// TIA Portal V15.1 export
// export: Created 2024-05-17T05:38:44.1667821Z, ExportSetting WithDefaults, DisplayName Totally Integrated Automation Portal, DisplayVersion V15.1 Update 5, DisplayName TIA Portal Openness, DisplayVersion V15.1 Update 5, DisplayName SINAMICS Startdrive Advanced, DisplayVersion V15.1, DisplayName G130, G150, S120, S150, SINAMICS MV, S210, DisplayVersion V15.1, DisplayName G110M, G120, G120C, G120D, G120P, DisplayVersion V15.1, DisplayName STEP 7 Professional, DisplayVersion V15.1 Update 5, DisplayName STEP 7 Safety, DisplayVersion V15.1, DisplayName WinCC Professional, DisplayVersion V15.1 Update 5, DisplayName SIMATIC Visualization Architect, DisplayVersion V15.1
FUNCTION_BLOCK "LGBVIDSChangeVEMData"   // FB6633, SCL
TITLE = LGBVIDSChangeVEMData
{ S7_Optimized_Access := 'FALSE' }
VERSION : 0.1
// stored: AutoNumber false, IsIECCheckEnabled false, SetENOAutomatically False, UDAEnableTagReadback false
   VAR_INPUT
      I_StartChangeVEMData { ExternalAccessible := 'False'; ExternalVisible := 'False'; ExternalWritable := 'False'} : Bool;   // Start command for coupling / Start command
      I_DataModeManEn { ExternalAccessible := 'False'; ExternalVisible := 'False'; ExternalWritable := 'False'} : Bool;   // Data mode manual - enable
   END_VAR
   VAR_OUTPUT
      O_DataModeAuto { ExternalAccessible := 'False'; ExternalVisible := 'False'; ExternalWritable := 'False'} : Bool;   // Couple or decouple in automatic mode / Data mode - Automatic
      O_DataModeMan { ExternalAccessible := 'False'; ExternalVisible := 'False'; ExternalWritable := 'False'} : Bool;   // Data mode - Manual
      O_Busy { ExternalAccessible := 'False'; ExternalVisible := 'False'; ExternalWritable := 'False'} : Bool;   // Busy
      O_Status { ExternalAccessible := 'False'; ExternalVisible := 'False'; ExternalWritable := 'False'} : Int;   // Status / Status (< 0 : fault, 0:No status, 1:Success, >0:Busy)
      O_Alarm { ExternalAccessible := 'False'; ExternalVisible := 'False'; ExternalWritable := 'False'} : Bool;   // Alarm
   END_VAR
   VAR_IN_OUT
      IO_VIDS : "VIDS";   // VIDS internal record
      IO_VEMData : "VEMData";   // VEM data
      IO_VEMDataChange : "VEMData";   // VEM data to be changed
      IO_CarrierCargoStatus : "VIDSCarrierCargoStatus";   // Carrier cargo status (Fixed layout)
      IO_CarrierCargoStatusChange : "VIDSCarrierCargoStatus";   // Carrier cargo status to be changed(Fixed layout)
      IO_BodyCargoStatus : "VIDSBodyCargoStatusGB";   // Body cargo status (Fixed layout)
      IO_BodyCargoStatusChange : "VIDSBodyCargoStatusGB";   // Body cargo status to be changed(Fixed layout)
      IO_WorkStatus : "VIDSWorkStatus";   // Work status(Fixed layout)
      IO_WorkStatusChange : "VIDSWorkStatus";   // Work status to be changed(Fixed layout)
      IO_EquipmentWork : "VIDSEquipment";
      IO_EquipmentWorkChange : "VIDSEquipment";
      IO_EquipmentWorkDone : "VIDSEquipment";
      IO_EquipmentWorkDoneChange : "VIDSEquipment";
      IO_Alarm : "Alarm";   // Alarm
      H_ChangeVEMData : "H_GBVIDSChangeVEMData";   // HMI interface
      H_HMI : "H_HMI";   // Icon animation
   END_VAR
   VAR DB_SPECIFIC
      RetVal { ExternalAccessible := 'False'; ExternalVisible := 'False'; ExternalWritable := 'False'} : Int;
      StartChangeVEMDataPls { ExternalAccessible := 'False'; ExternalVisible := 'False'; ExternalWritable := 'False'} : Bool;
      btnConfirmPls { ExternalAccessible := 'False'; ExternalVisible := 'False'; ExternalWritable := 'False'} : Bool;
      btnEditPls { ExternalAccessible := 'False'; ExternalVisible := 'False'; ExternalWritable := 'False'} : Bool;
      DataModeAuto { ExternalAccessible := 'False'; ExternalVisible := 'False'; ExternalWritable := 'False'} : Bool;   // Couple or decouple in automode
      DataModeAutoPls { ExternalAccessible := 'False'; ExternalVisible := 'False'; ExternalWritable := 'False'} : Bool;
      DataModeMan { ExternalAccessible := 'False'; ExternalVisible := 'False'; ExternalWritable := 'False'} : Bool;
      DataModeManPls { ExternalAccessible := 'False'; ExternalVisible := 'False'; ExternalWritable := 'False'} : Bool;
      DataModeMem { ExternalAccessible := 'False'; ExternalVisible := 'False'; ExternalWritable := 'False'} : Int;
      DataModeEdit { ExternalAccessible := 'False'; ExternalVisible := 'False'; ExternalWritable := 'False'} : Bool;
      DataModeChanged { ExternalAccessible := 'False'; ExternalVisible := 'False'; ExternalWritable := 'False'} : Bool;
      BeginReqPlsAuto { ExternalAccessible := 'False'; ExternalVisible := 'False'; ExternalWritable := 'False'} : Bool;
      BeginReqPlsMan { ExternalAccessible := 'False'; ExternalVisible := 'False'; ExternalWritable := 'False'} : Bool;
      SerializePos { ExternalAccessible := 'False'; ExternalVisible := 'False'; ExternalWritable := 'False'} : DInt;
      DeSerializePos { ExternalAccessible := 'False'; ExternalVisible := 'False'; ExternalWritable := 'False'} : DInt;
      VEMDataChangeMem { ExternalAccessible := 'False'; ExternalVisible := 'False'; ExternalWritable := 'False'; S7_SetPoint := 'True'} : "VEMData";
      VEMDataChangeMemArray { ExternalAccessible := 'False'; ExternalVisible := 'False'; ExternalWritable := 'False'} : Array[0..255] of Byte;
      Busy { ExternalAccessible := 'False'; ExternalVisible := 'False'; ExternalWritable := 'False'} : Bool;
      btnDataModeAutoColour { ExternalAccessible := 'False'; ExternalVisible := 'False'; ExternalWritable := 'False'} : Word;
      btnDataModeManColour { ExternalAccessible := 'False'; ExternalVisible := 'False'; ExternalWritable := 'False'} : Word;
      CarrierID { ExternalAccessible := 'False'; ExternalVisible := 'False'; ExternalWritable := 'False'} : DWord;
      CarrierIDValid { ExternalAccessible := 'False'; ExternalVisible := 'False'; ExternalWritable := 'False'} : Bool;
      CarrierIDMem { ExternalAccessible := 'False'; ExternalVisible := 'False'; ExternalWritable := 'False'} : DWord;   // Memory of CarrierID at begin request
      TagID { ExternalAccessible := 'False'; ExternalVisible := 'False'; ExternalWritable := 'False'} : DWord;
      TagIDValid { ExternalAccessible := 'False'; ExternalVisible := 'False'; ExternalWritable := 'False'} : Bool;
      TagIDMem { ExternalAccessible := 'False'; ExternalVisible := 'False'; ExternalWritable := 'False'} : DWord;
      BodyNbr { ExternalAccessible := 'False'; ExternalVisible := 'False'; ExternalWritable := 'False'} : DWord;
      BodyNbrValid { ExternalAccessible := 'False'; ExternalVisible := 'False'; ExternalWritable := 'False'} : Bool;
      BodyNbrMem { ExternalAccessible := 'False'; ExternalVisible := 'False'; ExternalWritable := 'False'} : DWord;
      MixNbr { ExternalAccessible := 'False'; ExternalVisible := 'False'; ExternalWritable := 'False'} : DWord;
      MixNbrValid { ExternalAccessible := 'False'; ExternalVisible := 'False'; ExternalWritable := 'False'} : Bool;
      MixNbrMem { ExternalAccessible := 'False'; ExternalVisible := 'False'; ExternalWritable := 'False'} : DWord;
      DataValid { ExternalAccessible := 'False'; ExternalVisible := 'False'; ExternalWritable := 'False'} : Bool;
      VEMDataValidPls { ExternalAccessible := 'False'; ExternalVisible := 'False'; ExternalWritable := 'False'} : Bool;
      InputDataValidAuto { ExternalAccessible := 'False'; ExternalVisible := 'False'; ExternalWritable := 'False'} : Bool;
      InputDataValidMan { ExternalAccessible := 'False'; ExternalVisible := 'False'; ExternalWritable := 'False'} : Bool;
      DataNotValid { ExternalAccessible := 'False'; ExternalVisible := 'False'; ExternalWritable := 'False'} : Bool;
      BeginPlsModeAuto { ExternalAccessible := 'False'; ExternalVisible := 'False'; ExternalWritable := 'False'} : Bool;   // Pulse of begin in auto mode
      BeginPlsModeManTagId { ExternalAccessible := 'False'; ExternalVisible := 'False'; ExternalWritable := 'False'} : Bool;   // Pulse of begin in manual mode
      BeginReqPls { ExternalAccessible := 'False'; ExternalVisible := 'False'; ExternalWritable := 'False'} : Bool;   // Pulse of begin request
      TagIdModeManMem { ExternalAccessible := 'False'; ExternalVisible := 'False'; ExternalWritable := 'False'} : DWord;   // Memorised TagId in manual mode
      Alarm { ExternalAccessible := 'False'; ExternalVisible := 'False'; ExternalWritable := 'False'} : Bool;   // Alarm
      ChangedRcvDataAlarm { ExternalAccessible := 'False'; ExternalVisible := 'False'; ExternalWritable := 'False'} : Bool;   // Alarm received data has chnged after request
      CoupleAlarm { ExternalAccessible := 'False'; ExternalVisible := 'False'; ExternalWritable := 'False'} : Bool;   // Alarm couple or decouple NOK
      Status { ExternalAccessible := 'False'; ExternalVisible := 'False'; ExternalWritable := 'False'} : Int;   // Status
      btnEditVisible { ExternalAccessible := 'False'; ExternalVisible := 'False'; ExternalWritable := 'False'} : Word;
      btnEditEnable { ExternalAccessible := 'False'; ExternalVisible := 'False'; ExternalWritable := 'False'} : Word;
      btnConfirmVisible { ExternalAccessible := 'False'; ExternalVisible := 'False'; ExternalWritable := 'False'} : Word;
      btnConfirmEnable { ExternalAccessible := 'False'; ExternalVisible := 'False'; ExternalWritable := 'False'} : Word;
      msgDataValidVisible { ExternalAccessible := 'False'; ExternalVisible := 'False'; ExternalWritable := 'False'} : Word;   // HMI - Couple/Decouple OK
      msgDataNotValidVisible { ExternalAccessible := 'False'; ExternalVisible := 'False'; ExternalWritable := 'False'} : Word;   // HMI - Couple/Decouple OK
      msgPartPresVisible { ExternalAccessible := 'False'; ExternalVisible := 'False'; ExternalWritable := 'False'} : Word;
      msgVEMDataCarrierVisible { ExternalAccessible := 'False'; ExternalVisible := 'False'; ExternalWritable := 'False'} : Word;
      msgVEMDataBodyVisible { ExternalAccessible := 'False'; ExternalVisible := 'False'; ExternalWritable := 'False'} : Word;
      txtCarrierIDVisible { ExternalAccessible := 'False'; ExternalVisible := 'False'; ExternalWritable := 'False'} : Word;
      txtCarrierIDEnable { ExternalAccessible := 'False'; ExternalVisible := 'False'; ExternalWritable := 'False'} : Word;
      txtCarrierIDColour { ExternalAccessible := 'False'; ExternalVisible := 'False'; ExternalWritable := 'False'} : Word;
      txtCarrierIDValid { ExternalAccessible := 'False'; ExternalVisible := 'False'; ExternalWritable := 'False'} : Bool;
      txtTagIDVisible { ExternalAccessible := 'False'; ExternalVisible := 'False'; ExternalWritable := 'False'} : Word;
      txtTagIDEnable { ExternalAccessible := 'False'; ExternalVisible := 'False'; ExternalWritable := 'False'} : Word;
      txtTagIDColour { ExternalAccessible := 'False'; ExternalVisible := 'False'; ExternalWritable := 'False'} : Word;
      txtTagIDValid { ExternalAccessible := 'False'; ExternalVisible := 'False'; ExternalWritable := 'False'} : Bool;
      txtMixNbrVisible { ExternalAccessible := 'False'; ExternalVisible := 'False'; ExternalWritable := 'False'} : Word;
      txtMixNbrEnable { ExternalAccessible := 'False'; ExternalVisible := 'False'; ExternalWritable := 'False'} : Word;
      txtMixNbrColour { ExternalAccessible := 'False'; ExternalVisible := 'False'; ExternalWritable := 'False'} : Word;
      txtMixNbrValid { ExternalAccessible := 'False'; ExternalVisible := 'False'; ExternalWritable := 'False'} : Bool;
      txtdestinationChangeVisible { ExternalAccessible := 'False'; ExternalVisible := 'False'; ExternalWritable := 'False'} : Word;
      txtdestinationChangeEnable { ExternalAccessible := 'False'; ExternalVisible := 'False'; ExternalWritable := 'False'} : Word;
      txtPlcProgramNumberChangeVisible { ExternalAccessible := 'False'; ExternalVisible := 'False'; ExternalWritable := 'False'} : Word;
      txtPlcProgramNumberChangeEnable { ExternalAccessible := 'False'; ExternalVisible := 'False'; ExternalWritable := 'False'} : Word;
      txtBodyNbrVisible { ExternalAccessible := 'False'; ExternalVisible := 'False'; ExternalWritable := 'False'} : Word;
      txtBodyNbrEnable { ExternalAccessible := 'False'; ExternalVisible := 'False'; ExternalWritable := 'False'} : Word;
      txtBodyNbrColour { ExternalAccessible := 'False'; ExternalVisible := 'False'; ExternalWritable := 'False'} : Word;
      txtBodyNbrValid { ExternalAccessible := 'False'; ExternalVisible := 'False'; ExternalWritable := 'False'} : Bool;
      txtSeqNbrChangeVisible { ExternalAccessible := 'False'; ExternalVisible := 'False'; ExternalWritable := 'False'} : Word;
      txtSeqNbrChangeEnable { ExternalAccessible := 'False'; ExternalVisible := 'False'; ExternalWritable := 'False'} : Word;
      txtRoutingChangeVisible { ExternalAccessible := 'False'; ExternalVisible := 'False'; ExternalWritable := 'False'} : Word;
      txtRoutingChangeEnable { ExternalAccessible := 'False'; ExternalVisible := 'False'; ExternalWritable := 'False'} : Word;
      txtWorkUntilChangeVisible { ExternalAccessible := 'False'; ExternalVisible := 'False'; ExternalWritable := 'False'} : Word;
      txtWorkUntilChangeEnable { ExternalAccessible := 'False'; ExternalVisible := 'False'; ExternalWritable := 'False'} : Word;
      txtBegWorkAfterChangeVisible { ExternalAccessible := 'False'; ExternalVisible := 'False'; ExternalWritable := 'False'} : Word;
      txtBegWorkAfterChangeEnable { ExternalAccessible := 'False'; ExternalVisible := 'False'; ExternalWritable := 'False'} : Word;
      selBodyCargoStatusChangeVisible { ExternalAccessible := 'False'; ExternalVisible := 'False'; ExternalWritable := 'False'} : Word;
      selBodyCargoStatusChangeEnable { ExternalAccessible := 'False'; ExternalVisible := 'False'; ExternalWritable := 'False'} : Word;
      selCarrierCargoStatusChangeVisible { ExternalAccessible := 'False'; ExternalVisible := 'False'; ExternalWritable := 'False'} : Word;
      selCarrierCargoStatusChangeEnable { ExternalAccessible := 'False'; ExternalVisible := 'False'; ExternalWritable := 'False'} : Word;
      selWorkStatusChangeVisible { ExternalAccessible := 'False'; ExternalVisible := 'False'; ExternalWritable := 'False'} : Word;
      selWorkStatusChangeEnable { ExternalAccessible := 'False'; ExternalVisible := 'False'; ExternalWritable := 'False'} : Word;
      selEquipmentWorkVisible { ExternalAccessible := 'False'; ExternalVisible := 'False'; ExternalWritable := 'False'} : Word;
      selEquipmentWorkEnable { ExternalAccessible := 'False'; ExternalVisible := 'False'; ExternalWritable := 'False'} : Word;
      selEquipmentWorkDoneVisible { ExternalAccessible := 'False'; ExternalVisible := 'False'; ExternalWritable := 'False'} : Word;
      selEquipmentWorkDoneEnable { ExternalAccessible := 'False'; ExternalVisible := 'False'; ExternalWritable := 'False'} : Word;
      IconColour { ExternalAccessible := 'False'; ExternalVisible := 'False'; ExternalWritable := 'False'} : Word;
      tempDWORDArray { ExternalAccessible := 'False'; ExternalVisible := 'False'; ExternalWritable := 'False'} : Array[0..31] of Bool;
   END_VAR
   VAR
      _DataModeManPls { ExternalAccessible := 'False'; ExternalVisible := 'False'; ExternalWritable := 'False'; S7_SetPoint := 'True'} : R_TRIG;
      _DataModeAutoPls { ExternalAccessible := 'False'; ExternalVisible := 'False'; ExternalWritable := 'False'; S7_SetPoint := 'True'} : R_TRIG;
      _btnConfirmPls { ExternalAccessible := 'False'; ExternalVisible := 'False'; ExternalWritable := 'False'; S7_SetPoint := 'True'} : R_TRIG;
      _btnEditPls { ExternalAccessible := 'False'; ExternalVisible := 'False'; ExternalWritable := 'False'; S7_SetPoint := 'True'} : R_TRIG;
      _VEMDataValidPls { ExternalAccessible := 'False'; ExternalVisible := 'False'; ExternalWritable := 'False'; S7_SetPoint := 'True'} : R_TRIG;
      _StartChangeVEMDataPls { ExternalAccessible := 'False'; ExternalVisible := 'False'; ExternalWritable := 'False'; S7_SetPoint := 'True'} : R_TRIG;
   END_VAR
   VAR DB_SPECIFIC
      _CoupleBeginOvTime { ExternalAccessible := 'False'; ExternalVisible := 'False'; ExternalWritable := 'False'; S7_SetPoint := 'True'} : TOF_TIME;
   END_VAR
   VAR
      _CoupleBeginWaitDonePls { ExternalAccessible := 'False'; ExternalVisible := 'False'; ExternalWritable := 'False'; S7_SetPoint := 'True'} : F_TRIG;
   END_VAR
   VAR DB_SPECIFIC
      _DeoupleBeginOvTime { ExternalAccessible := 'False'; ExternalVisible := 'False'; ExternalWritable := 'False'; S7_SetPoint := 'True'} : TOF_TIME;
   END_VAR
   VAR
      _DecoupleBeginWaitDonePls { ExternalAccessible := 'False'; ExternalVisible := 'False'; ExternalWritable := 'False'; S7_SetPoint := 'True'} : F_TRIG;
   END_VAR
   VAR_TEMP
      tempBool : Bool;
   END_VAR
   VAR CONSTANT
      STATUS_OK : Int := 1;
      STATUS_COUPLE_REQ : Int := 107;
      STATUS_COUPLE_RUNNING : Int := 207;
      STATUS_DECOUPLE_REQ : Int := 108;
      STATUS_DECOUPLE_RUNNING : Int := 208;
      OFF : Word := 2#0000000000000000;
      ON : Word := 2#0000000000000001;
      VISIBLE : Word := 2#0000000000000001;
      ENABLE : Word := 2#0000000000000010;
      COLOUR_DEFAULT : Word := 2#0000000000000000;
      COLOUR_RED : Word := 2#0000000000010000;
      COLOUR_GREEN : Word := 2#0000000000100000;
      COLOUR_BLUE : Word := 2#0000000001000000;
      COLOUR_WHITE : Word := 2#0000000010000000;
      CMD_CHANGE_DATA : DWord := 2001;
   END_VAR
BEGIN
   (******************************************************************************************
    Changelog

       21W29D3 18:00H 
       - New module

    List of authors

       Company : Volvo Cars Gent
       Name    : Christophe Staal
       E-mail  : christophe.staal@volvocars.com
       Tel.    : +32 470 34 60 98

    Description

       This module allows to change VEM data commonly used in B-shop

    ******************************************************************************)

   //Start change VEM data - Create pulse on edge
   #_StartChangeVEMDataPls(CLK := #I_StartChangeVEMData,
                   Q => #StartChangeVEMDataPls);

   //Button Confirm - Create pulse on edge
   #_btnConfirmPls(CLK := #H_ChangeVEMData.H_btnConfirm=#ON,
                   Q => #btnConfirmPls);

   //Button Edit - Create pulse on edge
   #_btnEditPls(CLK := #H_ChangeVEMData.H_btnEdit = #ON,
                Q => #btnEditPls);

   #_VEMDataValidPls(CLK := #IO_VIDS.VEMDataValid,
                Q => #VEMDataValidPls);

   (******************************************************************************)
   (* Data mode - Automatic                                                      *)
   (******************************************************************************)

   //Data mode selected  - No mode, select auto
      IF (#H_ChangeVEMData.H_selDataMode < 1) OR (#H_ChangeVEMData.H_selDataMode > 3) OR NOT #IO_VIDS.PartPres OR NOT #I_DataModeManEn THEN
          #H_ChangeVEMData.H_selDataMode := 1;
   END_IF;

   #DataModeAuto := #H_ChangeVEMData.H_selDataMode = 1;

   (******************************************************************************)
   (* Data mode - Manual                                                         *)
   (******************************************************************************)

   //Data mode MANUAL
   #DataModeMan := (#H_ChangeVEMData.H_selDataMode = 2);

   //Data mode changed
   #DataModeChanged := #H_ChangeVEMData.H_selDataMode <> #DataModeMem;
   #DataModeMem := #H_ChangeVEMData.H_selDataMode;

   (******************************************************************************)
   (* Data mode - Edit                                                           *)
   (******************************************************************************)

   IF #DataModeMan AND #btnEditPls THEN
       #DataModeEdit := TRUE;
   END_IF;

   (******************************************************************************)
   (* Update on VEM data valid                                                   *)
   (******************************************************************************)

   //Body Cargo status - update
   "LDWordToBit"(I_DWord:=#IO_VEMData.BodyCargoStatus,
                 O_0=>#IO_BodyCargoStatus.OK,
                 O_1=>#IO_BodyCargoStatus.NOK,
                 O_2=>#IO_BodyCargoStatus.Production,
                 O_3=>#IO_BodyCargoStatus.Test,
                 O_4=>#IO_BodyCargoStatus.Measurement,
                 O_5=>#IO_BodyCargoStatus.Scrap,
                 O_6=>#tempBool,
                 O_7=>#tempBool,
                 O_8=>#IO_BodyCargoStatus.Inspection,
                 O_9=>#tempBool,
                 O_10=>#IO_BodyCargoStatus.NoPriorityFlowDecisionByPLC,
                 O_11=>#IO_BodyCargoStatus.BodyCanGoTo5thCrane,
                 O_12=>#IO_BodyCargoStatus.BodyMustGoTo5thCrane,
                 O_13=>#IO_BodyCargoStatus.BodyCanNotGoTo5thCrane,
                 O_14=>#tempBool,
                 O_15=>#tempBool,
                 O_16=>#tempBool,
                 O_17=>#tempBool,
                 O_18=>#tempBool,
                 O_19=>#tempBool,
                 O_20=>#IO_BodyCargoStatus.BodyBufferFull,
                 O_21=>#IO_BodyCargoStatus.OvenBodyTC1Oven1,
                 O_22=>#IO_BodyCargoStatus.OvenBodyTC1Oven2,
                 O_23=>#IO_BodyCargoStatus.OvenBodyTC2Oven1,
                 O_24=>#IO_BodyCargoStatus.OvenBodyTC2Oven2,
                 O_25=>#IO_BodyCargoStatus.TestBodyTC1,
                 O_26=>#IO_BodyCargoStatus.TestBodyTC2,
                 O_27=>#tempBool,
                 O_28=>#tempBool,
                 O_29=>#tempBool,
                 O_30=>#tempBool,
                 O_31=>#IO_BodyCargoStatus.ExitWaterTestBody);

   //Carrier Cargo status - update
   "LDWordToBit"(I_DWord := #IO_VEMData.CarrierCargoStatus,
                 O_0 => #IO_CarrierCargoStatus.OK,
                 O_1 => #IO_CarrierCargoStatus.NOK,
                 O_2 => #IO_CarrierCargoStatus.Test,
                 O_3 => #IO_CarrierCargoStatus.Maint,
                 O_4 => #IO_CarrierCargoStatus.PrevMaint,
                 O_5 => #IO_CarrierCargoStatus.Loaded,
                 O_6 => #IO_CarrierCargoStatus.Job1,
                 O_7 => #IO_CarrierCargoStatus.Job2,
                 O_8 => #IO_CarrierCargoStatus.Job3,
                 O_9 => #tempBool,
                 O_10 => #tempBool,
                 O_11 => #tempBool,
                 O_12 => #tempBool,
                 O_13 => #tempBool,
                 O_14 => #tempBool,
                 O_15 => #tempBool,
                 O_16 => #tempBool,
                 O_17 => #tempBool,
                 O_18 => #tempBool,
                 O_19 => #tempBool,
                 O_20 => #tempBool,
                 O_21 => #tempBool,
                 O_22 => #tempBool,
                 O_23 => #tempBool,
                 O_24 => #tempBool,
                 O_25 => #tempBool,
                 O_26 => #tempBool,
                 O_27 => #tempBool,
                 O_28 => #tempBool,
                 O_29 => #tempBool,
                 O_30 => #tempBool,
                 O_31 => #tempBool);

   //Work status - update
   "LDWordToBit"(I_DWord := #IO_VEMData.WorkStatus,
                 O_0 => #IO_WorkStatus.Work,
                 O_1 => #IO_WorkStatus.NoWork,
                 O_2 => #IO_WorkStatus.BackupWork,
                 O_3 => #IO_WorkStatus.StopBefore,
                 O_4 => #IO_WorkStatus.StopAfter,
                 O_5 => #IO_WorkStatus.Quality,
                 O_6 => #tempBool,
                 O_7 => #tempBool,
                 O_8 => #tempBool,
                 O_9 => #tempBool,
                 O_10 => #tempBool,
                 O_11 => #tempBool,
                 O_12 => #tempBool,
                 O_13 => #tempBool,
                 O_14 => #tempBool,
                 O_15 => #tempBool,
                 O_16 => #tempBool,
                 O_17 => #tempBool,
                 O_18 => #tempBool,
                 O_19 => #tempBool,
                 O_20 => #tempBool,
                 O_21 => #tempBool,
                 O_22 => #tempBool,
                 O_23 => #tempBool,
                 O_24 => #tempBool,
                 O_25 => #tempBool,
                 O_26 => #tempBool,
                 O_27 => #tempBool,
                 O_28 => #tempBool,
                 O_29 => #tempBool,
                 O_30 => #tempBool,
                 O_31 => #tempBool);

   //Equipment Work - update
   "LDWordToBit"(I_DWord := #IO_VEMData.EquipmentWork,
                 O_0 => #IO_EquipmentWork.Bit[0],
                 O_1 => #IO_EquipmentWork.Bit[1],
                 O_2 => #IO_EquipmentWork.Bit[2],
                 O_3 => #IO_EquipmentWork.Bit[3],
                 O_4 => #IO_EquipmentWork.Bit[4],
                 O_5 => #IO_EquipmentWork.Bit[5],
                 O_6 => #IO_EquipmentWork.Bit[6],
                 O_7 => #IO_EquipmentWork.Bit[7],
                 O_8 => #IO_EquipmentWork.Bit[8],
                 O_9 => #IO_EquipmentWork.Bit[9],
                 O_10 => #IO_EquipmentWork.Bit[10],
                 O_11 => #IO_EquipmentWork.Bit[11],
                 O_12 => #IO_EquipmentWork.Bit[12],
                 O_13 => #IO_EquipmentWork.Bit[13],
                 O_14 => #IO_EquipmentWork.Bit[14],
                 O_15 => #IO_EquipmentWork.Bit[15],
                 O_16 => #IO_EquipmentWork.Bit[16],
                 O_17 => #IO_EquipmentWork.Bit[17],
                 O_18 => #IO_EquipmentWork.Bit[18],
                 O_19 => #IO_EquipmentWork.Bit[19],
                 O_20 => #IO_EquipmentWork.Bit[20],
                 O_21 => #IO_EquipmentWork.Bit[21],
                 O_22 => #IO_EquipmentWork.Bit[22],
                 O_23 => #IO_EquipmentWork.Bit[23],
                 O_24 => #IO_EquipmentWork.Bit[24],
                 O_25 => #IO_EquipmentWork.Bit[25],
                 O_26 => #IO_EquipmentWork.Bit[26],
                 O_27 => #IO_EquipmentWork.Bit[27],
                 O_28 => #IO_EquipmentWork.Bit[28],
                 O_29 => #IO_EquipmentWork.Bit[29],
                 O_30 => #IO_EquipmentWork.Bit[30],
                 O_31 => #IO_EquipmentWork.Bit[31]);

   //Equipment Work Done - update
   "LDWordToBit"(I_DWord := #IO_VEMData.EquipmentWorkDone,
                 O_0 => #IO_EquipmentWorkDone.Bit[0],
                 O_1 => #IO_EquipmentWorkDone.Bit[1],
                 O_2 => #IO_EquipmentWorkDone.Bit[2],
                 O_3 => #IO_EquipmentWorkDone.Bit[3],
                 O_4 => #IO_EquipmentWorkDone.Bit[4],
                 O_5 => #IO_EquipmentWorkDone.Bit[5],
                 O_6 => #IO_EquipmentWorkDone.Bit[6],
                 O_7 => #IO_EquipmentWorkDone.Bit[7],
                 O_8 => #IO_EquipmentWorkDone.Bit[8],
                 O_9 => #IO_EquipmentWorkDone.Bit[9],
                 O_10 => #IO_EquipmentWorkDone.Bit[10],
                 O_11 => #IO_EquipmentWorkDone.Bit[11],
                 O_12 => #IO_EquipmentWorkDone.Bit[12],
                 O_13 => #IO_EquipmentWorkDone.Bit[13],
                 O_14 => #IO_EquipmentWorkDone.Bit[14],
                 O_15 => #IO_EquipmentWorkDone.Bit[15],
                 O_16 => #IO_EquipmentWorkDone.Bit[16],
                 O_17 => #IO_EquipmentWorkDone.Bit[17],
                 O_18 => #IO_EquipmentWorkDone.Bit[18],
                 O_19 => #IO_EquipmentWorkDone.Bit[19],
                 O_20 => #IO_EquipmentWorkDone.Bit[20],
                 O_21 => #IO_EquipmentWorkDone.Bit[21],
                 O_22 => #IO_EquipmentWorkDone.Bit[22],
                 O_23 => #IO_EquipmentWorkDone.Bit[23],
                 O_24 => #IO_EquipmentWorkDone.Bit[24],
                 O_25 => #IO_EquipmentWorkDone.Bit[25],
                 O_26 => #IO_EquipmentWorkDone.Bit[26],
                 O_27 => #IO_EquipmentWorkDone.Bit[27],
                 O_28 => #IO_EquipmentWorkDone.Bit[28],
                 O_29 => #IO_EquipmentWorkDone.Bit[29],
                 O_30 => #IO_EquipmentWorkDone.Bit[30],
                 O_31 => #IO_EquipmentWorkDone.Bit[31]);

    IF #VEMDataValidPls THEN   

       //Body Cargo status change - update
     "LDWordToBit"(I_DWord := #IO_VEMDataChange.BodyCargoStatus,
                     O_0 => #IO_BodyCargoStatusChange.OK,
                     O_1 => #IO_BodyCargoStatusChange.NOK,
                     O_2 => #IO_BodyCargoStatusChange.Production,
                     O_3 => #IO_BodyCargoStatusChange.Test,
                     O_4 => #IO_BodyCargoStatusChange.Measurement,
                     O_5 => #IO_BodyCargoStatusChange.Scrap,
                     O_6 => #tempBool,
                     O_7 => #tempBool,
                     O_8 => #IO_BodyCargoStatusChange.Inspection,
                     O_9 => #tempBool,
                     O_10 => #IO_BodyCargoStatusChange.NoPriorityFlowDecisionByPLC,
                     O_11 => #IO_BodyCargoStatusChange.BodyCanGoTo5thCrane,
                     O_12 => #IO_BodyCargoStatusChange.BodyMustGoTo5thCrane,
                     O_13 => #IO_BodyCargoStatusChange.BodyCanNotGoTo5thCrane,
                     O_14 => #tempBool,
                     O_15 => #tempBool,
                     O_16 => #tempBool,
                     O_17 => #tempBool,
                     O_18 => #tempBool,
                     O_19 => #tempBool,
                     O_20 => #IO_BodyCargoStatusChange.BodyBufferFull,
                     O_21 => #IO_BodyCargoStatusChange.OvenBodyTC1Oven1,
                     O_22 => #IO_BodyCargoStatusChange.OvenBodyTC1Oven2,
                     O_23 => #IO_BodyCargoStatusChange.OvenBodyTC2Oven1,
                     O_24 => #IO_BodyCargoStatusChange.OvenBodyTC2Oven2,
                     O_25 => #IO_BodyCargoStatusChange.TestBodyTC1,
                     O_26 => #IO_BodyCargoStatusChange.TestBodyTC2,
                     O_27 => #tempBool,
                     O_28 => #tempBool,
                     O_29 => #tempBool,
                     O_30 => #tempBool,
                     O_31 => #IO_BodyCargoStatusChange.ExitWaterTestBody);

       //Carrier Cargo status change - update
       "LDWordToBit"(I_DWord := #IO_VEMDataChange.CarrierCargoStatus,
                     O_0 => #IO_CarrierCargoStatusChange.OK,
                     O_1 => #IO_CarrierCargoStatusChange.NOK,
                     O_2 => #IO_CarrierCargoStatusChange.Test,
                     O_3 => #IO_CarrierCargoStatusChange.Maint,
                     O_4 => #IO_CarrierCargoStatusChange.PrevMaint,
                     O_5 => #IO_CarrierCargoStatusChange.Loaded,
                     O_6 => #IO_CarrierCargoStatusChange.Job1,
                     O_7 => #IO_CarrierCargoStatusChange.Job2,
                     O_8 => #IO_CarrierCargoStatusChange.Job3,
                     O_9 => #tempBool,
                     O_10 => #tempBool,
                     O_11 => #tempBool,
                     O_12 => #tempBool,
                     O_13 => #tempBool,
                     O_14 => #tempBool,
                     O_15 => #tempBool,
                     O_16 => #tempBool,
                     O_17 => #tempBool,
                     O_18 => #tempBool,
                     O_19 => #tempBool,
                     O_20 => #tempBool,
                     O_21 => #tempBool,
                     O_22 => #tempBool,
                     O_23 => #tempBool,
                     O_24 => #tempBool,
                     O_25 => #tempBool,
                     O_26 => #tempBool,
                     O_27 => #tempBool,
                     O_28 => #tempBool,
                     O_29 => #tempBool,
                     O_30 => #tempBool,
                     O_31 => #tempBool);

       //Work status change - update
       "LDWordToBit"(I_DWord := #IO_VEMDataChange.WorkStatus,
                     O_0 => #IO_WorkStatusChange.Work,
                     O_1 => #IO_WorkStatusChange.NoWork,
                     O_2 => #IO_WorkStatusChange.BackupWork,
                     O_3 => #IO_WorkStatusChange.StopBefore,
                     O_4 => #IO_WorkStatusChange.StopAfter,
                     O_5 => #IO_WorkStatusChange.Quality,
                     O_6 => #tempBool,
                     O_7 => #tempBool,
                     O_8 => #tempBool,
                     O_9 => #tempBool,
                     O_10 => #tempBool,
                     O_11 => #tempBool,
                     O_12 => #tempBool,
                     O_13 => #tempBool,
                     O_14 => #tempBool,
                     O_15 => #tempBool,
                     O_16 => #tempBool,
                     O_17 => #tempBool,
                     O_18 => #tempBool,
                     O_19 => #tempBool,
                     O_20 => #tempBool,
                     O_21 => #tempBool,
                     O_22 => #tempBool,
                     O_23 => #tempBool,
                     O_24 => #tempBool,
                     O_25 => #tempBool,
                     O_26 => #tempBool,
                     O_27 => #tempBool,
                     O_28 => #tempBool,
                     O_29 => #tempBool,
                     O_30 => #tempBool,
                     O_31 => #tempBool);

       //Equipment Work change - update
       "LDWordToBit"(I_DWord := #IO_VEMDataChange.EquipmentWork,
                     O_0 => #IO_EquipmentWorkChange.Bit[0],
                     O_1 => #IO_EquipmentWorkChange.Bit[1],
                     O_2 => #IO_EquipmentWorkChange.Bit[2],
                     O_3 => #IO_EquipmentWorkChange.Bit[3],
                     O_4 => #IO_EquipmentWorkChange.Bit[4],
                     O_5 => #IO_EquipmentWorkChange.Bit[5],
                     O_6 => #IO_EquipmentWorkChange.Bit[6],
                     O_7 => #IO_EquipmentWorkChange.Bit[7],
                     O_8 => #IO_EquipmentWorkChange.Bit[8],
                     O_9 => #IO_EquipmentWorkChange.Bit[9],
                     O_10 => #IO_EquipmentWorkChange.Bit[10],
                     O_11 => #IO_EquipmentWorkChange.Bit[11],
                     O_12 => #IO_EquipmentWorkChange.Bit[12],
                     O_13 => #IO_EquipmentWorkChange.Bit[13],
                     O_14 => #IO_EquipmentWorkChange.Bit[14],
                     O_15 => #IO_EquipmentWorkChange.Bit[15],
                     O_16 => #IO_EquipmentWorkChange.Bit[16],
                     O_17 => #IO_EquipmentWorkChange.Bit[17],
                     O_18 => #IO_EquipmentWorkChange.Bit[18],
                     O_19 => #IO_EquipmentWorkChange.Bit[19],
                     O_20 => #IO_EquipmentWorkChange.Bit[20],
                     O_21 => #IO_EquipmentWorkChange.Bit[21],
                     O_22 => #IO_EquipmentWorkChange.Bit[22],
                     O_23 => #IO_EquipmentWorkChange.Bit[23],
                     O_24 => #IO_EquipmentWorkChange.Bit[24],
                     O_25 => #IO_EquipmentWorkChange.Bit[25],
                     O_26 => #IO_EquipmentWorkChange.Bit[26],
                     O_27 => #IO_EquipmentWorkChange.Bit[27],
                     O_28 => #IO_EquipmentWorkChange.Bit[28],
                     O_29 => #IO_EquipmentWorkChange.Bit[29],
                     O_30 => #IO_EquipmentWorkChange.Bit[30],
                     O_31 => #IO_EquipmentWorkChange.Bit[31]);

       //Equipment Work Done change - update
     "LDWordToBit"(I_DWord := #IO_VEMDataChange.EquipmentWorkDone,
                    O_0 => #IO_EquipmentWorkDoneChange.Bit[0],
                    O_1 => #IO_EquipmentWorkDoneChange.Bit[1],
                    O_2 => #IO_EquipmentWorkDoneChange.Bit[2],
                    O_3 => #IO_EquipmentWorkDoneChange.Bit[3],
                    O_4 => #IO_EquipmentWorkDoneChange.Bit[4],
                    O_5 => #IO_EquipmentWorkDoneChange.Bit[5],
                    O_6 => #IO_EquipmentWorkDoneChange.Bit[6],
                    O_7 => #IO_EquipmentWorkDoneChange.Bit[7],
                    O_8 => #IO_EquipmentWorkDoneChange.Bit[8],
                    O_9 => #IO_EquipmentWorkDoneChange.Bit[9],
                    O_10 => #IO_EquipmentWorkDoneChange.Bit[10],
                    O_11 => #IO_EquipmentWorkDoneChange.Bit[11],
                    O_12 => #IO_EquipmentWorkDoneChange.Bit[12],
                    O_13 => #IO_EquipmentWorkDoneChange.Bit[13],
                    O_14 => #IO_EquipmentWorkDoneChange.Bit[14],
                    O_15 => #IO_EquipmentWorkDoneChange.Bit[15],
                    O_16 => #IO_EquipmentWorkDoneChange.Bit[16],
                    O_17 => #IO_EquipmentWorkDoneChange.Bit[17],
                    O_18 => #IO_EquipmentWorkDoneChange.Bit[18],
                    O_19 => #IO_EquipmentWorkDoneChange.Bit[19],
                    O_20 => #IO_EquipmentWorkDoneChange.Bit[20],
                    O_21 => #IO_EquipmentWorkDoneChange.Bit[21],
                    O_22 => #IO_EquipmentWorkDoneChange.Bit[22],
                    O_23 => #IO_EquipmentWorkDoneChange.Bit[23],
                    O_24 => #IO_EquipmentWorkDoneChange.Bit[24],
                    O_25 => #IO_EquipmentWorkDoneChange.Bit[25],
                    O_26 => #IO_EquipmentWorkDoneChange.Bit[26],
                    O_27 => #IO_EquipmentWorkDoneChange.Bit[27],
                    O_28 => #IO_EquipmentWorkDoneChange.Bit[28],
                    O_29 => #IO_EquipmentWorkDoneChange.Bit[29],
                    O_30 => #IO_EquipmentWorkDoneChange.Bit[30],
                    O_31 => #IO_EquipmentWorkDoneChange.Bit[31]);

    END_IF;

   (******************************************************************************)
   (* Begin requests                                                             *)
   (******************************************************************************)

   //Begin request - Automatic mode
    #BeginReqPlsAuto := #StartChangeVEMDataPls AND #DataModeAuto AND #IO_VIDS.PartPres AND #IO_VIDS.VEMDataValid;

   IF #BeginReqPlsAuto THEN

       //Body Cargo status change - update
       "LBitToDword"(I_0:=#IO_BodyCargoStatusChange.OK,
                     I_1:=#IO_BodyCargoStatusChange.NOK,
                     I_2:=#IO_BodyCargoStatusChange.Production,
                     I_3:=#IO_BodyCargoStatusChange.Test,
                     I_4:=#IO_BodyCargoStatusChange.Measurement,
                     I_5:=#IO_BodyCargoStatusChange.Scrap,
                     I_6:=#tempBool,
                     I_7:=#tempBool,
                     I_8:=#IO_BodyCargoStatusChange.Inspection,
                     I_9:=#tempBool,
                     I_10:=#IO_BodyCargoStatusChange.NoPriorityFlowDecisionByPLC,
                     I_11:=#IO_BodyCargoStatusChange.BodyCanGoTo5thCrane,
                     I_12:=#IO_BodyCargoStatusChange.BodyMustGoTo5thCrane,
                     I_13:=#IO_BodyCargoStatusChange.BodyCanNotGoTo5thCrane,
                     I_14:=#tempBool,
                     I_15:=#tempBool,
                     I_16:=#tempBool,
                     I_17:=#tempBool,
                     I_18:=#tempBool,
                     I_19:=#tempBool,
                     I_20:=#IO_BodyCargoStatusChange.BodyBufferFull,
                     I_21:=#IO_BodyCargoStatusChange.OvenBodyTC1Oven1,
                     I_22:=#IO_BodyCargoStatusChange.OvenBodyTC1Oven2,
                     I_23:=#IO_BodyCargoStatusChange.OvenBodyTC2Oven1,
                     I_24:=#IO_BodyCargoStatusChange.OvenBodyTC2Oven2,
                     I_25:=#IO_BodyCargoStatusChange.TestBodyTC1,
                     I_26:=#IO_BodyCargoStatusChange.TestBodyTC2,
                     I_27:=#tempBool,
                     I_28:=#tempBool,
                     I_29:=#tempBool,
                     I_30:=#tempBool,
                     I_31:=#IO_BodyCargoStatusChange.ExitWaterTestBody,
                     O_DWord=>#IO_VEMDataChange.BodyCargoStatus);

       //Carrier Cargo status change - update
       "LBitToDword"(I_0 := #IO_CarrierCargoStatusChange.OK,
                     I_1 := #IO_CarrierCargoStatusChange.NOK,
                     I_2 := #IO_CarrierCargoStatusChange.Test,
                     I_3 := #IO_CarrierCargoStatusChange.Maint,
                     I_4 := #IO_CarrierCargoStatusChange.PrevMaint,
                     I_5 := #IO_CarrierCargoStatusChange.Loaded,
                     I_6 := #IO_CarrierCargoStatusChange.Job1,
                     I_7 := #IO_CarrierCargoStatusChange.Job2,
                     I_8 := #IO_CarrierCargoStatusChange.Job3,
                     I_9 := #tempBool,
                     I_10 := #tempBool,
                     I_11 := #tempBool,
                     I_12 := #tempBool,
                     I_13 := #tempBool,
                     I_14 := #tempBool,
                     I_15 := #tempBool,
                     I_16 := #tempBool,
                     I_17 := #tempBool,
                     I_18 := #tempBool,
                     I_19 := #tempBool,
                     I_20 := #tempBool,
                     I_21 := #tempBool,
                     I_22 := #tempBool,
                     I_23 := #tempBool,
                     I_24 := #tempBool,
                     I_25 := #tempBool,
                     I_26 := #tempBool,
                     I_27 := #tempBool,
                     I_28 := #tempBool,
                     I_29 := #tempBool,
                     I_30 := #tempBool,
                     I_31 := #tempBool,
                     O_DWord => #IO_VEMDataChange.CarrierCargoStatus);

       //Work status change - update
       "LBitToDword"(I_0 := #IO_WorkStatusChange.Work,
                     I_1 := #IO_WorkStatusChange.NoWork,
                     I_2 := #IO_WorkStatusChange.BackupWork,
                     I_3 := #IO_WorkStatusChange.StopBefore,
                     I_4 := #IO_WorkStatusChange.StopAfter,
                     I_5 := #IO_WorkStatusChange.Quality,
                     I_6 := #tempBool,
                     I_7 := #tempBool,
                     I_8 := #tempBool,
                     I_9 := #tempBool,
                     I_10 := #tempBool,
                     I_11 := #tempBool,
                     I_12 := #tempBool,
                     I_13 := #tempBool,
                     I_14 := #tempBool,
                     I_15 := #tempBool,
                     I_16 := #tempBool,
                     I_17 := #tempBool,
                     I_18 := #tempBool,
                     I_19 := #tempBool,
                     I_20 := #tempBool,
                     I_21 := #tempBool,
                     I_22 := #tempBool,
                     I_23 := #tempBool,
                     I_24 := #tempBool,
                     I_25 := #tempBool,
                     I_26 := #tempBool,
                     I_27 := #tempBool,
                     I_28 := #tempBool,
                     I_29 := #tempBool,
                     I_30 := #tempBool,
                     I_31 := #tempBool,
                     O_DWord => #IO_VEMDataChange.WorkStatus);

       //Equipment Work change - update
       "LBitToDword"(I_0 := #IO_EquipmentWorkChange.Bit[0],
                     I_1 := #IO_EquipmentWorkChange.Bit[1],
                     I_2 := #IO_EquipmentWorkChange.Bit[2],
                     I_3 := #IO_EquipmentWorkChange.Bit[3],
                     I_4 := #IO_EquipmentWorkChange.Bit[4],
                     I_5 := #IO_EquipmentWorkChange.Bit[5],
                     I_6 := #IO_EquipmentWorkChange.Bit[6],
                     I_7 := #IO_EquipmentWorkChange.Bit[7],
                     I_8 := #IO_EquipmentWorkChange.Bit[8],
                     I_9 := #IO_EquipmentWorkChange.Bit[9],
                     I_10 := #IO_EquipmentWorkChange.Bit[10],
                     I_11 := #IO_EquipmentWorkChange.Bit[11],
                     I_12 := #IO_EquipmentWorkChange.Bit[12],
                     I_13 := #IO_EquipmentWorkChange.Bit[13],
                     I_14 := #IO_EquipmentWorkChange.Bit[14],
                     I_15 := #IO_EquipmentWorkChange.Bit[15],
                     I_16 := #IO_EquipmentWorkChange.Bit[16],
                     I_17 := #IO_EquipmentWorkChange.Bit[17],
                     I_18 := #IO_EquipmentWorkChange.Bit[18],
                     I_19 := #IO_EquipmentWorkChange.Bit[19],
                     I_20 := #IO_EquipmentWorkChange.Bit[20],
                     I_21 := #IO_EquipmentWorkChange.Bit[21],
                     I_22 := #IO_EquipmentWorkChange.Bit[22],
                     I_23 := #IO_EquipmentWorkChange.Bit[23],
                     I_24 := #IO_EquipmentWorkChange.Bit[24],
                     I_25 := #IO_EquipmentWorkChange.Bit[25],
                     I_26 := #IO_EquipmentWorkChange.Bit[26],
                     I_27 := #IO_EquipmentWorkChange.Bit[27],
                     I_28 := #IO_EquipmentWorkChange.Bit[28],
                     I_29 := #IO_EquipmentWorkChange.Bit[29],
                     I_30 := #IO_EquipmentWorkChange.Bit[30],
                     I_31 := #IO_EquipmentWorkChange.Bit[31],
                     O_DWord => #IO_VEMDataChange.EquipmentWork);

       //Equipment Work Done change - update
       "LBitToDword"(I_0 := #IO_EquipmentWorkDoneChange.Bit[0],
                     I_1 := #IO_EquipmentWorkDoneChange.Bit[1],
                     I_2 := #IO_EquipmentWorkDoneChange.Bit[2],
                     I_3 := #IO_EquipmentWorkDoneChange.Bit[3],
                     I_4 := #IO_EquipmentWorkDoneChange.Bit[4],
                     I_5 := #IO_EquipmentWorkDoneChange.Bit[5],
                     I_6 := #IO_EquipmentWorkDoneChange.Bit[6],
                     I_7 := #IO_EquipmentWorkDoneChange.Bit[7],
                     I_8 := #IO_EquipmentWorkDoneChange.Bit[8],
                     I_9 := #IO_EquipmentWorkDoneChange.Bit[9],
                     I_10 := #IO_EquipmentWorkDoneChange.Bit[10],
                     I_11 := #IO_EquipmentWorkDoneChange.Bit[11],
                     I_12 := #IO_EquipmentWorkDoneChange.Bit[12],
                     I_13 := #IO_EquipmentWorkDoneChange.Bit[13],
                     I_14 := #IO_EquipmentWorkDoneChange.Bit[14],
                     I_15 := #IO_EquipmentWorkDoneChange.Bit[15],
                     I_16 := #IO_EquipmentWorkDoneChange.Bit[16],
                     I_17 := #IO_EquipmentWorkDoneChange.Bit[17],
                     I_18 := #IO_EquipmentWorkDoneChange.Bit[18],
                     I_19 := #IO_EquipmentWorkDoneChange.Bit[19],
                     I_20 := #IO_EquipmentWorkDoneChange.Bit[20],
                     I_21 := #IO_EquipmentWorkDoneChange.Bit[21],
                     I_22 := #IO_EquipmentWorkDoneChange.Bit[22],
                     I_23 := #IO_EquipmentWorkDoneChange.Bit[23],
                     I_24 := #IO_EquipmentWorkDoneChange.Bit[24],
                     I_25 := #IO_EquipmentWorkDoneChange.Bit[25],
                     I_26 := #IO_EquipmentWorkDoneChange.Bit[26],
                     I_27 := #IO_EquipmentWorkDoneChange.Bit[27],
                     I_28 := #IO_EquipmentWorkDoneChange.Bit[28],
                     I_29 := #IO_EquipmentWorkDoneChange.Bit[29],
                     I_30 := #IO_EquipmentWorkDoneChange.Bit[30],
                     I_31 := #IO_EquipmentWorkDoneChange.Bit[31],
                     O_DWord => #IO_VEMDataChange.EquipmentWorkDone);

   END_IF;

   //Begin request - Manual mode
   #BeginReqPlsMan := #DataModeEdit AND #btnConfirmPls AND #DataModeMan;

   IF #BeginReqPlsMan THEN
       //Update VEMDataChange with HMI fields
       #IO_VEMDataChange.BodyCargoStatus := #H_ChangeVEMData.H_selBodyCargoStatusChange;
       #IO_VEMDataChange.CarrierCargoStatus := #H_ChangeVEMData.H_selCarrierCargoStatusChange;
       #IO_VEMDataChange.WorkStatus := #H_ChangeVEMData.H_selWorkStatusChange;
       #IO_VEMDataChange.EquipmentWork := #H_ChangeVEMData.H_selEquipmentWorkChange;
       #IO_VEMDataChange.EquipmentWorkDone := #H_ChangeVEMData.H_selEquipmentWorkDoneChange;

       #IO_VEMDataChange.SequenceNumber := #H_ChangeVEMData.H_txtSeqNbrChange;
       #IO_VEMDataChange.Routing := #H_ChangeVEMData.H_txtRoutingChange;
       #IO_VEMDataChange.WorkUntil := #H_ChangeVEMData.H_txtWorkUntilChange;
       #IO_VEMDataChange.BegWorkAfter := #H_ChangeVEMData.H_txtBegWorkAfterChange;
       #IO_VEMDataChange.Destination := #H_ChangeVEMData.H_txtDestinationChange;
       #IO_VEMDataChange.PLCProgramNumber := #H_ChangeVEMData.H_txtPlcProgramNumberChange;

   END_IF;

   //Data mode edit - Off
   IF #DataModeChanged OR #BeginReqPlsMan THEN
       #DataModeEdit := FALSE;
   END_IF;

   //Memorize parameters
   IF #BeginReqPlsAuto OR #BeginReqPlsMan THEN
       #SerializePos := 0;
       #RetVal:=Serialize(SRC_VARIABLE:=#IO_VEMDataChange, DEST_ARRAY=>#VEMDataChangeMemArray, POS:=#SerializePos);
   END_IF;

   //Begin request - Summary
   #IO_VIDS.ChangeData.BeginReq := #BeginReqPlsAuto OR #BeginReqPlsMan;

   (******************************************************************************)
   (* Begin                                                                      *)
   (******************************************************************************)

   //Initialize parameters
   IF #IO_VIDS.ChangeData.OkBegin THEN
       #DeSerializePos := 0;
       #RetVal := Deserialize(SRC_ARRAY := #VEMDataChangeMemArray, DEST_VARIABLE => #IO_VIDS.VEMData, POS := #DeSerializePos);
       #IO_VIDS.VEMData.CommandCode := #CMD_CHANGE_DATA;
       #IO_VIDS.VEMData.SpecificDataLength := 0;      // Set SpecificDataLenght to ZERO
   END_IF;

   //Begin
   #IO_VIDS.ChangeData.Begin := #IO_VIDS.ChangeData.OkBegin;

   (******************************************************************************)
   (* Busy                                                                       *)
   (******************************************************************************)
   IF #IO_VIDS.ChangeData.Running THEN
       #Status := #IO_VIDS.ChangeData.Status;
       #Busy := TRUE;
   END_IF;

   (******************************************************************************)
   (* Finished                                                                   *)
   (******************************************************************************)

   IF #IO_VIDS.ChangeData.Finished THEN
       #Status := #IO_VIDS.ChangeData.Status;
       #Busy := False;
   END_IF;

   (******************************************************************************)
   (* Alarm                                                                      *)
   (******************************************************************************)

   #Alarm := (#Status < 0);

   "LAlarmSummary"(I_AlarmA:= "FALSE",
                   I_AlarmB:="FALSE",
                   I_AlarmC:= #Alarm,
                   I_AlarmD:="FALSE",
                   I_AlarmABCondition:="FALSE",
                   IO_Alarm:= #IO_Alarm,
                   C_UpperLevelHW:="FALSE",
                   C_UpperLevelSafety:="FALSE",
                   C_Safety:="FALSE",
                   C_Mechanic:="FALSE",
                   C_Transport:="FALSE",
                   C_Feature1:="FALSE",
                   C_Feature2:="FALSE",
                   C_Feature3:="FALSE");


   (******************************************************************************)
   (* Clear data                                                                 *)
   (******************************************************************************)
   IF #IO_VIDS.ChangeData.BeginReq OR #DataModeChanged OR NOT #IO_VIDS.PartPres THEN
       #DataValid := False;
       #DataNotValid := False;
       #Status := 0;
   END_IF;

   (******************************************************************************)
   (* Outputs                                                                    *)
   (******************************************************************************)

   #O_Busy := #Busy;
   #O_Alarm := #Alarm;
   #O_Status := #Status;
   #O_DataModeMan := #DataModeMan;
   #O_DataModeAuto := #DataModeAuto;

   (*******************************************************)
   (* HMI - Buttons                                       *)
   (*******************************************************)

   //HMI - Button Data mode automatic
   IF #DataModeAuto THEN
       #btnDataModeAutoColour := #COLOUR_GREEN;
   ELSE
       #btnDataModeAutoColour := #COLOUR_DEFAULT;
   END_IF;

   //HMI - Button Data mode manual
   IF #DataModeMan THEN
       #btnDataModeManColour := #COLOUR_BLUE;
   ELSE
       #btnDataModeManColour := #COLOUR_DEFAULT;
   END_IF;

   //HMI - Button Edit
   IF #DataModeMan AND NOT #DataModeEdit AND NOT #IO_VIDS.ChangeData.Running THEN
       #btnEditVisible := #VISIBLE;
       #btnEditEnable := #ENABLE;
   ELSE
       #btnEditVisible := #OFF;
       #btnEditEnable := #OFF;
   END_IF;

   //HMI - Button Confirm
   IF #DataModeEdit AND NOT #IO_VIDS.ChangeData.Running THEN
       #btnConfirmVisible := #VISIBLE;
       #btnConfirmEnable := #ENABLE;
   ELSE
       #btnConfirmVisible := #OFF;
       #btnConfirmEnable := #OFF;
   END_IF;

   (*******************************************************)
   (* HMI - Update text fields                            *)
   (*******************************************************)

   #H_ChangeVEMData.H_txtCarrierID := #IO_VEMData.CarrierID;
   #H_ChangeVEMData.H_txtBodyID := #IO_VEMData.BodyID;
   #H_ChangeVEMData.H_txtSeqNbr := #IO_VEMData.SequenceNumber;
   #H_ChangeVEMData.H_txtRouting := #IO_VEMData.Routing;
   #H_ChangeVEMData.H_txtWorkUntil := #IO_VEMData.WorkUntil;
   #H_ChangeVEMData.H_txtBegWorkAfter := #IO_VEMData.BegWorkAfter;
   #H_ChangeVEMData.H_txtDestination := #IO_VEMData.Destination;
   #H_ChangeVEMData.H_txtPlcProgramNumber := #IO_VEMData.PLCProgramNumber;
   #H_ChangeVEMData.H_txtPopId := #IO_VEMData.PopID;                  
   #H_ChangeVEMData.H_txtPopIdSuffix := #IO_VEMData.PopIDSuffix;
   #H_ChangeVEMData.H_txtPopType := #IO_VEMData.PopType;

   IF #VEMDataValidPls THEN
       #H_ChangeVEMData.H_txtSeqNbrChange := #IO_VEMData.SequenceNumber;
       #H_ChangeVEMData.H_txtRoutingChange := #IO_VEMData.Routing;
       #H_ChangeVEMData.H_txtWorkUntilChange := #IO_VEMData.WorkUntil;
       #H_ChangeVEMData.H_txtBegWorkAfterChange := #IO_VEMData.BegWorkAfter;
       #H_ChangeVEMData.H_txtDestinationChange := #IO_VEMData.Destination;
       #H_ChangeVEMData.H_txtPlcProgramNumberChange := #IO_VEMData.PLCProgramNumber;
   END_IF;

   //
   IF #DataModeEdit THEN
       #txtSeqNbrChangeVisible := #VISIBLE;
       #txtSeqNbrChangeEnable := #ENABLE;
       #txtRoutingChangeVisible := #VISIBLE;
       #txtRoutingChangeEnable :=  #ENABLE;
       #txtWorkUntilChangeVisible := #VISIBLE;
       #txtWorkUntilChangeEnable := #ENABLE;
       #txtBegWorkAfterChangeVisible  := #VISIBLE;
       #txtBegWorkAfterChangeEnable := #ENABLE;
       #txtdestinationChangeVisible := #VISIBLE;
       #txtdestinationChangeEnable := #ENABLE;
       #txtPlcProgramNumberChangeVisible := #VISIBLE;
       #txtPlcProgramNumberChangeEnable := #ENABLE;

   ELSE
       #txtSeqNbrChangeVisible := #OFF;
       #txtSeqNbrChangeEnable := #OFF;
       #txtRoutingChangeVisible := #OFF;
       #txtRoutingChangeEnable := #OFF;
       #txtWorkUntilChangeVisible := #OFF;
       #txtWorkUntilChangeEnable := #OFF;
       #txtBegWorkAfterChangeVisible := #OFF;
       #txtBegWorkAfterChangeEnable := #OFF;
       #txtdestinationChangeVisible := #OFF;
       #txtdestinationChangeEnable := #OFF;
       #txtPlcProgramNumberChangeVisible := #OFF;
       #txtPlcProgramNumberChangeEnable := #OFF;

   END_IF;

   (*******************************************************)
   (* HMI - Messages                                      *)
   (*******************************************************)

   //HMI - Message part present
   IF #IO_VIDS.PartPres THEN
       #msgPartPresVisible := #VISIBLE;
   ELSE
       #msgPartPresVisible := #OFF;
   END_IF;

   //HMI - Message data valid, not valid
   IF #IO_VIDS.VEMDataValid THEN
       #msgDataValidVisible := #VISIBLE;
   ELSIF #IO_VIDS.VEMDataNotValid THEN
       #msgDataNotValidVisible := #VISIBLE;
   ELSE
       #msgDataValidVisible := #OFF;
       #msgDataNotValidVisible := #OFF;
   END_IF;

   //Body or carrier data
   IF #IO_VIDS.IDType = 0 THEN
       #msgVEMDataBodyVisible := #VISIBLE;
       #msgVEMDataCarrierVisible := #OFF;
   ELSE
       #msgVEMDataBodyVisible := #OFF;
       #msgVEMDataCarrierVisible := #VISIBLE;
   END_IF;

   (*******************************************************)
   (* HMI - Selections                                    *)
   (*******************************************************)

   IF #VEMDataValidPls THEN
       #H_ChangeVEMData.H_selBodyCargoStatusChange := #IO_VEMData.BodyCargoStatus;
       #H_ChangeVEMData.H_selCarrierCargoStatusChange := #IO_VEMData.CarrierCargoStatus;
       #H_ChangeVEMData.H_selWorkStatusChange := #IO_VEMData.WorkStatus;
       #H_ChangeVEMData.H_selEquipmentWorkChange := #IO_VEMData.EquipmentWork;
       #H_ChangeVEMData.H_selEquipmentWorkDoneChange := #IO_VEMData.EquipmentWorkDone;
   END_IF;

   //
   IF #DataModeEdit THEN
       #selBodyCargoStatusChangeVisible := #VISIBLE;
       #selBodyCargoStatusChangeEnable := #ENABLE;
       #selCarrierCargoStatusChangeVisible := #VISIBLE;
       #selCarrierCargoStatusChangeEnable := #ENABLE;
       #selWorkStatusChangeVisible := #VISIBLE;
       #selWorkStatusChangeEnable := #ENABLE;
       #selEquipmentWorkVisible := #VISIBLE;
       #selEquipmentWorkEnable := #ENABLE;
       #selEquipmentWorkDoneVisible := #VISIBLE;
       #selEquipmentWorkDoneEnable := #ENABLE;
   ELSE
       #selBodyCargoStatusChangeVisible := #OFF;
       #selBodyCargoStatusChangeEnable := #OFF;
       #selCarrierCargoStatusChangeVisible := #OFF;
       #selCarrierCargoStatusChangeEnable := #OFF;
       #selWorkStatusChangeVisible := #OFF;
       #selWorkStatusChangeEnable := #OFF;
       #selEquipmentWorkVisible := #OFF;
       #selEquipmentWorkEnable := #OFF;
       #selEquipmentWorkDoneVisible := #OFF;
       #selEquipmentWorkDoneEnable := #OFF;
   END_IF;

   (*******************************************************)
   (* HMI - Indications                                   *)
   (*******************************************************)

   #H_ChangeVEMData.H_indBodyCargoStatus := #IO_VEMData.BodyCargoStatus;
   #H_ChangeVEMData.H_indCarrierCargoStatus := #IO_VEMData.CarrierCargoStatus;
   #H_ChangeVEMData.H_indWorkStatus := #IO_VEMData.WorkStatus;
   #H_ChangeVEMData.H_indEquipmentWork := #IO_VEMData.EquipmentWork;
   #H_ChangeVEMData.H_indEquipmentWorkDone := #IO_VEMData.EquipmentWorkDone;

   (*******************************************************)
   (* HMI - Animations summary                            *)
   (*******************************************************)

   //Buttons
   #H_ChangeVEMData.H_btnDataModeAutoAnim := #btnDataModeAutoColour;
   #H_ChangeVEMData.H_btnDataModeManAnim := #btnDataModeManColour;
   #H_ChangeVEMData.H_btnEditAnim := #btnEditVisible OR #btnEditEnable;
   #H_ChangeVEMData.H_btnConfirmAnim := #btnConfirmVisible OR #btnConfirmEnable;

   //Text fields
   #H_ChangeVEMData.H_txtSeqNbrChangeAnim := #txtSeqNbrChangeVisible OR #txtSeqNbrChangeEnable;
   #H_ChangeVEMData.H_txtRoutingChangeAnim := #txtRoutingChangeVisible OR #txtRoutingChangeEnable;
   #H_ChangeVEMData.H_txtWorkUntilChangeAnim := #txtWorkUntilChangeVisible OR #txtWorkUntilChangeEnable;
   #H_ChangeVEMData.H_txtBegWorkAfterChangeAnim := #txtBegWorkAfterChangeVisible OR #txtBegWorkAfterChangeEnable;
   #H_ChangeVEMData.H_txtDestinationChangeAnim := #txtdestinationChangeVisible OR #txtdestinationChangeEnable;
   #H_ChangeVEMData.H_txtPlcProgramNumberAnim := #txtPlcProgramNumberChangeVisible OR #txtPlcProgramNumberChangeEnable;

   //Selections
   #H_ChangeVEMData.H_selBodyCargoStatusChangeAnim := #selBodyCargoStatusChangeVisible OR #selBodyCargoStatusChangeEnable;
   #H_ChangeVEMData.H_selCarrierCargoStatusChangeAnim := #selCarrierCargoStatusChangeVisible OR #selCarrierCargoStatusChangeEnable;
   #H_ChangeVEMData.H_selWorkStatusChangeAnim := #selWorkStatusChangeVisible OR #selWorkStatusChangeEnable;
   #H_ChangeVEMData.H_selEquipmentWorkChangeAnim := #selEquipmentWorkVisible OR #selEquipmentWorkEnable;
   #H_ChangeVEMData.H_selEquipmentWorkDoneChangeAnim := #selEquipmentWorkDoneVisible OR #selEquipmentWorkDoneEnable;

   //Messages
   #H_ChangeVEMData.H_msgPartPresAnim := #msgPartPresVisible;
   #H_ChangeVEMData.H_msgVEMDataValidAnim := #msgDataValidVisible;
   #H_ChangeVEMData.H_msgVEMDataNotValidAnim := #msgDataNotValidVisible;
   #H_ChangeVEMData.H_msgStatus := #Status;

   (******************************************************************************)
   (* HMI - Reset buttons                                                        *)
   (******************************************************************************)

   #H_ChangeVEMData.H_btnEdit := #OFF;
   #H_ChangeVEMData.H_btnConfirm := #OFF;

   (******************************************************************************)
   (* Status To HMI word - Anim                                                  *)
   (******************************************************************************)
   "LBitToDword"(I_0:=#I_DataModeManEn,
                 I_1:=#DataModeEdit,
                 I_2:="FALSE",
                 I_3:="FALSE",
                 I_4:="FALSE",
                 I_5:="FALSE",
                 I_6:="FALSE",
                 I_7:="FALSE",
                 I_8:="FALSE",
                 I_9:="FALSE",
                 I_10:="FALSE",
                 I_11:="FALSE",
                 I_12:="FALSE",
                 I_13:="FALSE",
                 I_14:="FALSE",
                 I_15:="FALSE",
                 I_16:="FALSE",
                 I_17:="FALSE",
                 I_18:="FALSE",
                 I_19:="FALSE",
                 I_20:="FALSE",
                 I_21:="FALSE",
                 I_22:="FALSE",
                 I_23:="FALSE",
                 I_24:="FALSE",
                 I_25:="FALSE",
                 I_26:="FALSE",
                 I_27:="FALSE",
                 I_28:="FALSE",
                 I_29:="FALSE",
                 I_30:="FALSE",
                 I_31:="FALSE",
                 O_DWord=>#H_ChangeVEMData.H_Anim);

   (******************************************************************************)
   (* Status To HMI word - IAnim                                                 *)
   (******************************************************************************)
   //*** Machine #Status - Indication *** TO HMI - Icon animation
   "LIAnimDWord"(I_SetPos := "FALSE",
                 I_ResetPos := "FALSE",
                 I_Active := #Status = 2,
                 I_Visible := "FALSE",
                 I_OutOfUse := "FALSE",
                 I_IntlkSet := "FALSE",
                 I_IntlkReset := "FALSE",
                 I_IntlkSetAlm := "FALSE",
                 I_IntlkResetAlm := "FALSE",
                 I_ManualMode := #DataModeMan,
                 I_FncSelInHMI := "FALSE",
                 I_AnySelected := "FALSE",
                 I_AlarmA := "FALSE",
                 I_AlarmB := "FALSE",
                 I_AlarmC := #DataNotValid OR  #Status < 0,
                 I_AlarmD := "FALSE",
                 I_SafetyOk := "FALSE",
                 I_Service:="TRUE",
                 I_Spare1:="FALSE",
                 I_Spare2:="FALSE",
                 I_Spare3:="FALSE",
                 I_Spare4:="FALSE",
                 I_Spare5:="FALSE",
                 I_Spare6:="FALSE",
                 I_Spare7:="FALSE",
                 I_Spare8:="FALSE",
                 I_Spare9:="FALSE",
                 I_Spare10:="FALSE",
                 I_Spare11:="FALSE",
                 I_Spare12:="FALSE",
                 I_Spare13:="FALSE",
                 I_Spare14:="FALSE",
                 H_IAnim => #H_HMI.H_IAnim);
END_FUNCTION_BLOCK
